{attribute 'qualified_only'}
VAR_GLOBAL
	Tags: AdsTagsParallelUnits;
END_VAR

(* stored: Version 1.1.0.1, ProductVersion 3.1.4024.6
   GVL ADS_ParallelUnits: Id {2fbc342d-b22a-416a-a986-781df2feba0f} *)
